TYPE ST_AlarmLifecycleState :
STRUCT
	Latched : BOOL;
	PreviousActive : BOOL;
	SeenThisCycle : BOOL;
	Alarm : ST_ExtAlarm;
END_STRUCT
END_TYPE

(* stored: Version 1.1.0.1, ProductVersion 3.1.4026.18
   DUT ST_AlarmLifecycleState: Id {711ede85-7607-43f2-a233-271f83f2a8dc} *)
